FUNCTION_BLOCK Validation
VAR
	errors : ARRAY[0..GVL.maxMessages] OF STRING_5K;
	warnings : ARRAY[0..GVL.maxMessages] OF STRING_5K;

	tempErrors : ARRAY[0..GVL.maxMessages] OF STRING_5K;
	tempWarnings : ARRAY[0..GVL.maxMessages] OF STRING_5K;
	numErr : INT;
	numWarn : INT;
	
	bundleExists : BOOL;
		
	dbCheckStep : (CONNECT, READY, EXECUTE, FINISH);
	validationStep : (CHECK_EXISTING_BUNDLE, VALIDATE_DATA, FINISH_VALIDATION);
END_VAR

CASE validationStep OF
	CHECK_EXISTING_BUNDLE:
		IF checkExistingBundles() THEN
			validationStep := VALIDATE_DATA;
		END_IF
	
	VALIDATE_DATA:
		validateGeneralData(); //general data
		validateProcess(); //required processing
		validateMaterials(); //recipe
		
		validationStep := FINISH_VALIDATION;
		
	FINISH_VALIDATION: //copy temp to ADS and clear temp
		MEMCPY(ADR(errors), ADR(tempErrors), SIZEOF(errors));
		MEMCPY(ADR(warnings), ADR(tempWarnings), SIZEOF(warnings));
		
		MEMSET(ADR(tempErrors), 0, SIZEOF(tempErrors));
		MEMSET(ADR(tempWarnings), 0, SIZEOF(tempWarnings));
		numErr := 0;
		numWarn := 0;
		
		validationStep := CHECK_EXISTING_BUNDLE;
END_CASE

METHOD checkExistingBundles : BOOL
VAR_INST
	fbSQLCommand : FB_SQLCommandEvt(sNetID := '', tTimeout := T#5S);
	fbSQLDatabase : FB_SQLDatabaseEvt(sNetID := '', tTimeout := T#5S);
	fbSQLResult: FB_SQLResultEvt(sNetID := '', tTimeout := T#5S);
	
	
	cmd : ARRAY[0..2] OF STRING_5K;
	query : STRING_5K;
	tcMessage : I_TcMessage;
	existingID : STRING;
END_VAR
CASE dbCheckStep OF
	CONNECT:
		IF fbSQLDatabase.Connect(1) THEN
			IF NOT fbSqlDatabase.bError THEN
				dbCheckStep := READY;
			END_IF
		END_IF
		
	READY:
		IF fbSQLDatabase.CreateCmd(ADR(fbSQLCommand)) THEN
			dbCheckStep := EXECUTE;
		END_IF
	
	EXECUTE:
		cmd[0] := 'SELECT BundleID FROM "Bundle Data - Prototype" WHERE BundleID = $'';
		cmd[1] := TO_STRING(BundleData.id);
		cmd[2] := '$'';
		query := ConcatStrings(cmd, '', '', '');
		
		IF fbSQLCommand.ExecuteDataReturn(ADR(query), SIZEOF(query), ADR(fbSqlResult)) THEN
			dbCheckStep := FINISH;
		END_IF
		
	FINISH:
		fbSqlResult.Read(0, 1, ADR(existingID), SIZEOF(existingID), TRUE, FALSE);
		IF BundleData.id = existingID THEN
			bundleExists := TRUE;
		ELSE
			bundleExists := FALSE;
		END_IF
		IF fbSQLDatabase.Disconnect() THEN
			fbSqlResult.Release();
			checkExistingBundles := TRUE;
			dbCheckStep := CONNECT;
		END_IF
END_CASE
END_METHOD

{attribute 'TcRpcEnable'}
METHOD validateCardboard : BOOL
VAR_INST
	i : DINT;
END_VAR
FOR i:=0 TO GVL.maxMaterials BY 1 DO
	IF i > 0 THEN
		IF
			StrapWrapRecipe.Cardboard[i].position = StrapWrapRecipe.Cardboard[i-1].position 
			AND
			NOT(StrapWrapRecipe.Cardboard[i].position = 0 OR StrapWrapRecipe.Cardboard[i-1].position = 0)
		THEN
			tempWarnings[numWarn] := 'Cardboard: duplicate position';
			numWarn := numWarn + 1;
		END_IF
	END_IF
END_FOR
END_METHOD

{attribute 'TcRpcEnable'}
METHOD validateChipboard : BOOL
VAR_INST
	i : DINT;
END_VAR
FOR i:=0 TO GVL.maxMaterials BY 1 DO
	IF i > 0 THEN
		IF 
			StrapWrapRecipe.Chipboard[i].position = StrapWrapRecipe.Chipboard[i-1].position 
			AND
			NOT(StrapWrapRecipe.Chipboard[i].position = 0 OR StrapWrapRecipe.Chipboard[i-1].position = 0)
		THEN
			tempWarnings[numWarn] := 'Chipboard: duplicate position';
			numWarn := numWarn + 1;
		END_IF
	END_IF
END_FOR
END_METHOD

{attribute 'TcRpcEnable'}
METHOD validateCornerGuard : BOOL
VAR_INST
	i : DINT;
END_VAR
FOR i:=0 TO GVL.maxMaterials BY 1 DO
	IF i > 0 THEN
		IF 
			StrapWrapRecipe.CornerGuard[i].position = StrapWrapRecipe.CornerGuard[i-1].position 
			AND
			NOT(StrapWrapRecipe.CornerGuard[i].position = 0 OR StrapWrapRecipe.CornerGuard[i-1].position = 0)
		THEN
			tempWarnings[numWarn] := 'Corner Guard: duplicate position';
			numWarn := numWarn + 1;
		END_IF
	END_IF
END_FOR
END_METHOD

METHOD validateGeneralData : BOOL
IF BundleData.id = '' THEN //bundle id
	tempErrors[numErr] := 'ID missing';
	numErr := numErr + 1;
ELSIF BundleData.id <> '' AND bundleExists THEN
	tempWarnings[numWarn] := 'Bundle with entered ID already exists, proceeding will overwrite the existing recipe';
	numWarn := numWarn + 1;
END_IF

IF BundleData.weight = 0 THEN
	tempErrors[numErr] := 'Bundle weight missing';
	numErr := numErr + 1;
END_IF
IF BundleData.length = 0 OR BundleData.height = 0 OR BundleData.width = 0 THEN
	tempErrors[numErr] := 'Bundle dimension(s) missing';
	numErr := numErr + 1;
END_IF
IF BundleData.pieces = 0 OR BundleData.layers = 0 OR BundleData.piecesPerLayer = 0 THEN
	tempErrors[numErr] := 'Bundle layer dimension(s) missing';
	numErr := numErr + 1;
END_IF

IF Extrusiondata.extrusionWeight = 0 THEN
	tempErrors[numErr] := 'Extrusion weight missing';
	numErr := numErr + 1;
END_IF

IF Extrusiondata.extrusionHeight = 0 OR Extrusiondata.extrusionWidth = 0 THEN
	tempErrors[numErr] := 'Extrusion dimension(s) missing';
	numErr := numErr + 1;
END_IF
END_METHOD

{attribute 'TcRpcEnable'}
METHOD validateMaterials : BOOL
VAR_INST
	//fbSQLCommand : FB_SQLCommandEvt(sNetID := '', tTimeout := T#5S);
	//fbSQLDatabase : FB_SQLDatabaseEvt (sNetID := '', tTimeout := T#5S);
	//fbSQLResult: FB_SQLResultEvt(sNetID:='', tTimeout:=T#5S);
	
	
	
	
	//sqlResult : FB_SQLResult;
	
END_VAR

validatePaper();
validateCardboard();
validateCornerGuard();
validateChipboard();
validateWoodBunk();
END_METHOD

{attribute 'TcRpcEnable'}
METHOD validatePaper : BOOL
VAR_INST
	i : DINT;
END_VAR
FOR i:=0 TO GVL.maxMaterials BY 1 DO
	IF StrapWrapRecipe.TopPaper[i].start = 0 AND StrapWrapRecipe.TopPaper[i].end = 0 THEN //unused entry, do nothing and skip
		CONTINUE;
	END_IF
	
	IF StrapWrapRecipe.TopPaper[i].start >= StrapWrapRecipe.TopPaper[i].end THEN //invalid interval where start > end
		tempErrors[numErr] := 'Paper (Top): Start position must be less than end position';
		numErr := numErr + 1;
	END_IF
	
	IF i > 0 THEN
		IF StrapWrapRecipe.TopPaper[i].start < StrapWrapRecipe.TopPaper[i-1].end AND StrapWrapRecipe.TopPaper[i-1].end > 0 THEN //overlaps
			tempWarnings[numWarn] := 'Paper (Top): Overlapping segments';
			numWarn := numWarn + 1;
		ELSIF StrapWrapRecipe.TopPaper[i].start = StrapWrapRecipe.TopPaper[i-1].end AND StrapWrapRecipe.TopPaper[i-1].end > 0 THEN //adjacency
			tempWarnings[numWarn] := 'Paper (Top): Adjacent segments';
			numWarn := numWarn + 1;
		END_IF
	END_IF
END_FOR

FOR i:=0 TO GVL.maxMaterials BY 1 DO
	IF StrapWrapRecipe.LeftPaper[i].start = 0 AND StrapWrapRecipe.LeftPaper[i].end = 0 THEN //unused entry, do nothing and skip
		CONTINUE;
	END_IF
	
	IF StrapWrapRecipe.LeftPaper[i].start >= StrapWrapRecipe.LeftPaper[i].end THEN //invalid interval where start > end
		tempErrors[numErr] := 'Paper (Left): Start position must be less than end position';
		numErr := numErr + 1;
	END_IF
	
	IF i > 0 THEN
		IF StrapWrapRecipe.LeftPaper[i].start < StrapWrapRecipe.LeftPaper[i-1].end AND StrapWrapRecipe.LeftPaper[i-1].end > 0 THEN //overlaps
			tempWarnings[numWarn] := 'Paper (Left): Overlapping intervals, ignore if this is intended';
			numWarn := numWarn + 1;
		ELSIF StrapWrapRecipe.LeftPaper[i].start = StrapWrapRecipe.LeftPaper[i-1].end AND StrapWrapRecipe.LeftPaper[i-1].end > 0 THEN //adjacency
			tempWarnings[numWarn] := 'Paper (Left): Adjacent intervals can connected, ignore if this is intended';
			numWarn := numWarn + 1;
		END_IF
	END_IF
END_FOR

FOR i:=0 TO GVL.maxMaterials BY 1 DO
	IF StrapWrapRecipe.RightPaper[i].start = 0 AND StrapWrapRecipe.RightPaper[i].end = 0 THEN //unused entry, do nothing and skip
		CONTINUE;
	END_IF
	
	IF StrapWrapRecipe.RightPaper[i].start >= StrapWrapRecipe.RightPaper[i].end THEN //invalid interval where start > end
		tempErrors[numErr] := 'Paper (Right): Start position must be less than end position';
		numErr := numErr + 1;
	END_IF
	
	IF i > 0 THEN
		IF StrapWrapRecipe.RightPaper[i].start < StrapWrapRecipe.RightPaper[i-1].end AND StrapWrapRecipe.RightPaper[i-1].end > 0 THEN //overlaps
			tempWarnings[numWarn] := 'Paper (Right): Overlapping intervals, ignore if this is intended';
			numWarn := numWarn + 1;
		ELSIF StrapWrapRecipe.RightPaper[i].start = StrapWrapRecipe.RightPaper[i-1].end AND StrapWrapRecipe.RightPaper[i-1].end > 0 THEN //adjacency
			tempWarnings[numWarn] := 'Paper (Right): Adjacent intervals can connected, ignore if this is intended';
			numWarn := numWarn + 1;
		END_IF
	END_IF
END_FOR

FOR i:=0 TO GVL.maxMaterials BY 1 DO
	IF StrapWrapRecipe.BottomPaper[i].start = 0 AND StrapWrapRecipe.BottomPaper[i].end = 0 THEN //unused entry, do nothing and skip
		CONTINUE;
	END_IF
	
	IF StrapWrapRecipe.BottomPaper[i].start >= StrapWrapRecipe.BottomPaper[i].end THEN //invalid interval where start > end
		tempErrors[numErr] := 'Paper (Bottom): Start position must be less than end position';
		numErr := numErr + 1;
	END_IF
	
	IF i > 0 THEN
		IF StrapWrapRecipe.BottomPaper[i].start < StrapWrapRecipe.BottomPaper[i-1].end AND StrapWrapRecipe.BottomPaper[i-1].end > 0 THEN //overlaps
			tempWarnings[numWarn] := 'Paper (Bottom): Overlapping segments';
			numWarn := numWarn + 1;
		ELSIF StrapWrapRecipe.BottomPaper[i].start = StrapWrapRecipe.BottomPaper[i-1].end AND StrapWrapRecipe.BottomPaper[i-1].end > 0 THEN //adjacency
			tempWarnings[numWarn] := 'Paper (Bottom): Adjacent segments';
			numWarn := numWarn + 1;
		END_IF
	END_IF
END_FOR
END_METHOD

METHOD validateProcess : BOOL
VAR_INPUT
END_VAR
IF ( //if recipe exists but auto/manual strap and wrap is not selected
	StrapWrapRecipe.TopPaper[0].end > 0 OR 
	StrapWrapRecipe.LeftPaper[0].end > 0 OR 
	StrapWrapRecipe.RightPaper[0].end > 0 OR
	StrapWrapRecipe.BottomPaper[0].end > 0 OR 
	
	StrapWrapRecipe.Cardboard[0].top <> '' OR 
	StrapWrapRecipe.Cardboard[0].left <> '' OR 
	StrapWrapRecipe.Cardboard[0].right <> '' OR 
	StrapWrapRecipe.Cardboard[0].bottom <> '' OR 
	
	StrapWrapRecipe.Cardboard[0].topLeft <> '' OR 
	StrapWrapRecipe.Cardboard[0].topRight <> '' OR 
	StrapWrapRecipe.Cardboard[0].bottomLeft <> '' OR 
	StrapWrapRecipe.Cardboard[0].bottomRight <> '' OR 
	
	StrapWrapRecipe.CornerGuard[0].topLeft <> '' OR 
	StrapWrapRecipe.CornerGuard[0].topRight <> '' OR 
	StrapWrapRecipe.CornerGuard[0].bottomLeft <> '' OR 
	StrapWrapRecipe.CornerGuard[0].bottomRight <> '' OR 
	
	StrapWrapRecipe.Chipboard[0].top <> '' OR 
	StrapWrapRecipe.Chipboard[0].left <> '' OR 
	StrapWrapRecipe.Chipboard[0].right <> '' OR 
	StrapWrapRecipe.Chipboard[0].Bottom <> '' OR 

	StrapWrapRecipe.WoodBunk[0].top <> '' OR 
	StrapWrapRecipe.WoodBunk[0].left <> '' OR 
	StrapWrapRecipe.WoodBunk[0].right <> '' OR 
	StrapWrapRecipe.WoodBunk[0].Bottom <> '')
THEN
	IF NOT BundleData.requiredProcessing[BundleData.AUTO_SS] AND NOT BundleData.requiredProcessing[BundleData.MANUAL_SS] THEN
		tempErrors[numErr] := 'Recipe exists but strap and wrap processes are not selected (Auto/Manual Strap and Wrap)';
		numErr := numErr + 1;
	END_IF
ELSE //no recipe exists but auto/manual strap and wrap is selected
	IF BundleData.requiredProcessing[BundleData.AUTO_SS] OR BundleData.requiredProcessing[BundleData.MANUAL_SS] THEN
		tempWarnings[numWarn] := 'Strap and wrap processes are selected but there is no recipe, is this intended?';
		numWarn := numWarn + 1;
	END_IF
END_IF

	
IF //auto and manual strap/wrap are both selected
	(BundleData.requiredProcessing[BundleData.AUTO_RE] AND BundleData.requiredProcessing[BundleData.MANUAL_RE]) OR
	(BundleData.requiredProcessing[BundleData.AUTO_SS] AND BundleData.requiredProcessing[BundleData.MANUAL_SS])
THEN
	tempErrors[numErr] := 'Auto and Manual processes of the same type cannot be selected together';
	numErr := numErr + 1;
	
ELSIF //no processes selected
	NOT BundleData.requiredProcessing[BundleData.AUTO_RE] AND 
	NOT BundleData.requiredProcessing[BundleData.AUTO_SS] AND
	NOT BundleData.requiredProcessing[BundleData.MANUAL_RE] AND 
	NOT BundleData.requiredProcessing[BundleData.MANUAL_SS]
THEN
	tempWarnings[numWarn] := 'No processes are selected, is this intended?';
	numWarn := numWarn + 1;
END_IF
END_METHOD

{attribute 'TcRpcEnable'}
METHOD validateWoodBunk : BOOL
VAR_INST
	i : DINT;
END_VAR
FOR i:=0 TO GVL.maxMaterials BY 1 DO
	IF i > 0 THEN
		IF 
			StrapWrapRecipe.WoodBunk[i].position = StrapWrapRecipe.WoodBunk[i-1].position 
			AND
			NOT(StrapWrapRecipe.WoodBunk[i].position = 0 OR StrapWrapRecipe.WoodBunk[i-1].position = 0)
		THEN
			tempWarnings[numWarn] := 'Wood Bunk: duplicate position';
			numWarn := numWarn + 1;
		END_IF
	END_IF
END_FOR
END_METHOD

END_FUNCTION_BLOCK

(* stored: Version 1.1.0.1, ProductVersion 3.1.4024.11
   POU Validation: Id {2464cf26-8c9f-4fbe-9ea4-d9320ca9dedd}, SpecialFunc None
   Folder Validation Helpers: Id {336bab4d-dfe1-43cc-8122-3620813a0a71}
   Method checkExistingBundles: Id {11fec9c7-2dcd-4b8b-a43e-aec449f61511}
   Method validateCardboard: Id {2b3695ad-06b1-4918-a8a3-f03b87508814}
   Method validateChipboard: Id {85d71b23-c0e7-4dee-815a-c41b453aeaab}
   Method validateCornerGuard: Id {5130abb2-8880-4812-b2fe-bc561a83b061}
   Method validateGeneralData: Id {02e44bac-6aac-40e9-a641-9c054bdbaf32}
   Method validateMaterials: Id {1ae1a68e-dac5-4e97-8a19-d881f7d2bd32}
   Method validatePaper: Id {6e6d7d8a-4304-4b81-8399-c41f86090a25}
   Method validateProcess: Id {1f7c5baf-3a53-43c0-9455-37b7360ed8c7}
   Method validateWoodBunk: Id {02083b5d-e4d9-49ef-a36c-660d2366a08f} *)
